FUNCTION_BLOCK TimeTest (* Composite Function Block Type *)
  (* Standard: 61499-2 *)
  (* Version 0.0, 4/20/2016, DiM, nxtControl GmbH, template *)
  PACKAGE Main;
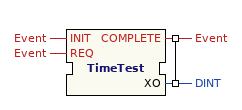
  EVENT_INPUT
    INIT; (* Initialization Request *)
    REQ; (* Normal Execution Request *)
  END_EVENT
  EVENT_OUTPUT
    COMPLETE WITH XO; (* Initialization Confirm *)
  END_EVENT
  VAR_OUTPUT
    XO : DINT; (* Output event qualifier *)
  END_VAR
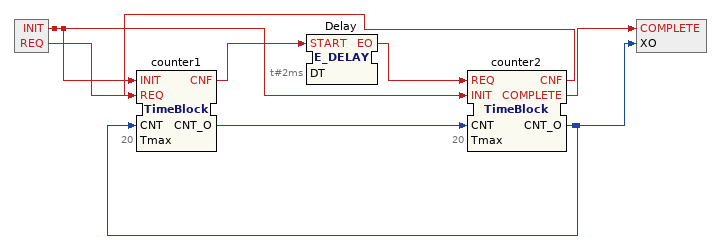
  FBS
    Delay : E_DELAY(DT := t#2ms);
    counter1 : TimeBlock(Tmax := 20);
    counter2 : TimeBlock(Tmax := 20);
  END_FBS
  EVENT_CONNECTIONS
    INIT TO counter1.INIT;
    counter1.CNF TO Delay.START;
    Delay.EO TO counter2.REQ;
    INIT TO counter2.INIT;
    REQ TO counter1.REQ;
    counter2.CNF TO counter1.REQ;
    counter2.COMPLETE TO COMPLETE;
  END_CONNECTIONS
  DATA_CONNECTIONS
    counter1.CNT_O TO counter2.CNT;
    counter2.CNT_O TO counter1.CNT;
    counter2.CNT_O TO XO;
  END_CONNECTIONS
END_FUNCTION_BLOCK
